# EPICS autosave request: support/ccd/1-10/ccdApp/Db/smartControl_settings.req
# FILE... smartControl_settings.req
$(P)$(R)debugLevel
file "smartControl_settings_axisX.req", P=$(P), R=$(R), AXIS=TTH
file "smartControl_settings_axisX.req", P=$(P), R=$(R), AXIS=OMEGA
file "smartControl_settings_axisX.req", P=$(P), R=$(R), AXIS=PHI
file "smartControl_settings_axisX.req", P=$(P), R=$(R), AXIS=KAPPA
